Universal Robots PolyScope program: BiBaZu_Continuous.urp

Program BiBaZu_Continuous (installation=default directory=/programs/usbdisk createdIn=5.12.3.1101619 lastSavedIn=5.12.3.1101619 robotSerialNumber=20225600150)
Calibrated DH parameters: a=[0.000094, -0.358471, -0.354967, -0.000026, 0.000038, 0]; d=[0.180831, -2593.499827, 2607.523833, -13.849973, 0.119817, 0.115619]; alpha=[1.570306, -0.000122, 0.004332, 1.569125, -1.569785, 0]; deltaTheta=[0, 0.723437, 5.729253, -0.169511, 0.000001, 0]
BeforeStart
  Script file BiBaZu_Continuous_Init.script
    | def BiBaZu_Continuous_Init():
    |   global angle = 0
    |   global last_command = read_input_integer_register(43)
    |   global active_command = last_command
    |   global command_valid = False
    |   global rotation_position = p[0, 0, 0, 0, 0, 0]
    |   write_output_integer_register(42, last_command)
    |   write_output_integer_register(43, 1)
    |   write_output_integer_register(41, 0)
    | end
    | 
    | BiBaZu_Continuous_Init()
  MoveJ speed 60 deg/s, acceleration 80 deg/s^2 (useActiveTCP=true) feature=Base
    Waypoint Rotation_Position: TCP in base x=-276.529 y=-617.246 z=308.214 mm, rx=0.4375 ry=1.1444 rz=-2.7623 rad; joints [-97.997, -121.173, -107.904, 271.738, -82.953, -161.379] deg
  Script file BiBaZu_Continuous_CapturePose.script
    | def BiBaZu_Continuous_CapturePose():
    |   global rotation_position = get_actual_tcp_pose()
    | end
    | 
    | BiBaZu_Continuous_CapturePose()
Robot Program (runOnlyOnce=false)
  angle := 0
  Script file BiBaZu_Continuous_Wait.script
    | def BiBaZu_Continuous_Wait():
    |   local command = read_input_integer_register(43)
    |   while command == last_command:
    |     sync()
    |     command = read_input_integer_register(43)
    |   end
    | 
    |   local requested_angle = read_input_integer_register(42)
    |   local valid = requested_angle >= 155 and requested_angle <= 210
    | 
    |   if valid:
    |     global angle = requested_angle
    |     global active_command = command
    |     global command_valid = True
    |     write_output_integer_register(43, 2)
    |   else:
    |     global angle = 0
    |     global command_valid = False
    |     global last_command = command
    |     write_output_integer_register(43, -1)
    |     write_output_integer_register(42, command)
    |   end
    | end
    | 
    | BiBaZu_Continuous_Wait()
  Script file BiBaZu_Continuous_Move.script
    | def BiBaZu_Continuous_Move():
    |   if command_valid:
    |     local target_rpy = [d2r(-45.0), d2r(angle / 10.0), d2r(-90.0)]
    |     local target_rotation = rpy2rotvec(target_rpy)
    |     local target_pose = p[rotation_position[0], rotation_position[1], rotation_position[2], target_rotation[0], target_rotation[1], target_rotation[2]]
    |     movel(target_pose, a=0.3, v=0.1)
    |   end
    | end
    | 
    | BiBaZu_Continuous_Move()
  Script file BiBaZu_Continuous_Ack.script
    | def BiBaZu_Continuous_Ack():
    |   if command_valid:
    |     write_output_integer_register(41, angle)
    |     write_output_integer_register(43, 3)
    |     write_output_integer_register(42, active_command)
    |     global last_command = active_command
    |     global command_valid = False
    |   end
    | end
    | 
    | BiBaZu_Continuous_Ack()
